// TwinCAT 3 PLC project Nestec
// libraries:
//   Tc2_ControllerToolbox,newest,Beckhoff Automation GmbH
//   Tc2_Standard,newest,Beckhoff Automation GmbH
//   Tc2_System,newest,Beckhoff Automation GmbH
//   Tc2_Utilities,newest,Beckhoff Automation GmbH
//   Tc3_Interfaces,3.3.0.0,Beckhoff Automation GmbH
//   Tc3_Module,3.3.6.0,Beckhoff Automation GmbH
// project tree:
//   Global Variables/ Global_Constantes.TcGVL, Global_IOs.TcGVL, TwinCAT_Configuration.TcGVL, Variable_Configuration.TcGVL
//   / GlobalImagePool.TcIPO (not stored), GlobalTextList.TcGTLO, Slow.TcTTO, Standard.TcTTO, Visualization Manager.TcVMO (not stored)
//   POUs/EMS/ EMS_Start.TcPOU
//   POUs/Flowrate management/ CALCULATE_FLOW.TcPOU, FLOWMETER.TcPOU
//   POUs/Functions/ PUMP_POWER.TcPOU, STATION_MODE.TcPOU
//   POUs/ MAIN.TcPOU
//   POUs/PC/ TO_PC.TcPOU
//   POUs/Tests/ getFlowrate.TcPOU, test.TcPOU, test_pressure.TcPOU, test_sonde_temp_G01.TcPOU, test_temp_G01.TcPOU, test_vacuum.TcPOU
//   Visualizations/ Visu1.TcVIS

CONFIGURATION Nestec
    RESOURCE PLC ON TwinCAT3
        TASK Slow(INTERVAL := T#100000us, PRIORITY := 21);
        TASK Standard(INTERVAL := T#10ms, PRIORITY := 20);
        PROGRAM CALCULATE_FLOW WITH Slow : CALCULATE_FLOW;
        PROGRAM MAIN WITH Standard : MAIN;
    END_RESOURCE
END_CONFIGURATION

// ---- Global Variables/Global_Constantes.TcGVL
{attribute 'Tc2GvlVarNames'}
VAR_GLOBAL


	R_BTN_S3: BOOL;



END_VAR

// ---- Global Variables/Global_IOs.TcGVL
{attribute 'Tc2GvlVarNames'}
VAR_GLOBAL

(**************************************
*
* PC variables 
*
***************************************)

(*FROM PC*)
	PC_ST1_PUMP_STATUS	:INT;(*0 OFF // 1 ON*)
	PC_ST2_PUMP_STATUS	:INT;
	PC_ST3_PUMP_STATUS	:INT;
	PC_ST4_PUMP_STATUS	:INT;

	PC_ST1_MODE			:INT;(*0 débit/pression // 1 pression max // 2 aspiration*)
	PC_ST2_MODE			:INT;
	PC_ST3_MODE			:INT;
	PC_ST4_MODE			:INT;

	PC_RESET_EMS			:BOOL; (*TO reset Emergency start*)

	PC_INIT					:BOOL;

(*TO PC*)
	PC_ST1_PRESSURE		:REAL;
	PC_ST2_PRESSURE		:REAL;
	PC_ST3_PRESSURE		:REAL;
	PC_ST4_PRESSURE		:REAL;

	PC_ST1_SUCTION		:REAL;
	PC_ST2_SUCTION		:REAL;
	PC_ST3_SUCTION		:REAL;
	PC_ST4_SUCTION		:REAL;

	PC_ST1_FLOWRATE		:REAL;
	PC_ST2_FLOWRATE		:REAL;
	PC_ST3_FLOWRATE		:REAL;
	PC_ST4_FLOWRATE		:REAL;

	PC_ST1_TEMP			:REAL;
	PC_ST2_TEMP			:REAL;
	PC_ST3_TEMP			:REAL;
	PC_ST4_TEMP			:REAL;

	PC_ST1_TEMP_ERROR	:BOOL;
	PC_ST2_TEMP_ERROR	:BOOL;
	PC_ST3_TEMP_ERROR	:BOOL;
	PC_ST4_TEMP_ERROR	:BOOL;

	PC_ST1_CURRENT		:REAL;
	PC_ST2_CURRENT		:REAL;
	PC_ST3_CURRENT		:REAL;
	PC_ST4_CURRENT		:REAL;

	PC_ST1_POWER			:REAL;
	PC_ST2_POWER			:REAL;
	PC_ST3_POWER			:REAL;
	PC_ST4_POWER			:REAL;

	PC_ST1_BTN			:BOOL;
	PC_ST2_BTN			:BOOL;
	PC_ST3_BTN			:BOOL;
	PC_ST4_BTN			:BOOL;

	PC_EMS_OK				:BOOL; (*EMS is SAFE*)






(**************************************
*
* EMERGECY STOP
*
***************************************)

	EMS_RESET		AT%Q*: BOOL;
	EMS_RUN		AT%Q*: BOOL;
	EMS_ACK 		AT%Q*: BOOL;

	EMS_FB_ERR	AT%I*: BOOL;
	EMS_COM_ERR	AT%I*: BOOL;
	EMS_OUT_ERR	AT%I*: BOOL;

	(*1: State RUN
	2: State STOP
	3: State SAFE
	4: State ERROR
	5: State RESET
	6: State START
	8: State DELAYOUT
	*)
	EMS_STATE		AT%I*:USINT;

	EMS_OK			AT%I*:BOOL;	(*Emergency stop is OK*)

(**************************************
*
* Inputs
*
***************************************)

	BTN_S3 AT%I*: BOOL;
	BTN_S4 AT%I*: BOOL;
	BTN_S5 AT%I*: BOOL;
	BTN_S6 AT%I*: BOOL;

	Weight_Station1 AT%I*:REAL;
	Weight_Station2 AT%I*:REAL;
	Weight_Station3 AT%I*:REAL;
	Weight_Station4 AT%I*:REAL;


	Temp_Station1 AT%I*:INT;
	Temp1_error   AT%I*:BOOL;
	Temp_Station2 AT%I*:INT;
	Temp2_error   AT%I*:BOOL;
	Temp_Station3 AT%I*:INT;
	Temp3_error   AT%I*:BOOL;
	Temp_Station4 AT%I*:INT;
	Temp4_error   AT%I*:BOOL;


	Vacuum_Station1 AT%I*:INT;
	Vacuum_Station2 AT%I*:INT;
	Vacuum_Station3 AT%I*:INT;
	Vacuum_Station4 AT%I*:INT;


	Pressure_Station1 AT%I*:INT;
	Pressure_Station2 AT%I*:INT;
	Pressure_Station3 AT%I*:INT;
	Pressure_Station4 AT%I*:INT;


	Temperature_entree_1 AT%I*:REAL;
	Temperature_entree_2 AT%I*:REAL;



(**************************************
*
* Outputs
*
***************************************)

	Alim_1 AT%Q*: BOOL;
	Alim_2 AT%Q*: BOOL;
	Alim_3 AT%Q*: BOOL;
	Alim_4 AT%Q*: BOOL;


	Mot_1 AT%Q*: BOOL;
	Mot_2 AT%Q*: BOOL;
	Mot_3 AT%Q*: BOOL;
	Mot_4 AT%Q*: BOOL;


	Solenoid_W13 AT%Q*: BOOL;
	Solenoid_W14 AT%Q*: BOOL;
	Solenoid_W15 AT%Q*: BOOL;
	Solenoid_W16 AT%Q*: BOOL;
	Solenoid_W17 AT%Q*: BOOL;
	Solenoid_W18 AT%Q*: BOOL;
	Solenoid_W19 AT%Q*: BOOL;
	Solenoid_W20 AT%Q*: BOOL;


	Light_H1 AT%Q*: BOOL;
	Light_H2 AT%Q*: BOOL;
	Light_H3 AT%Q*: BOOL;
	Light_H4 AT%Q*: BOOL;

(**************************************
*
* Multimeter IOs
*
***************************************)

	ST1_Multimeter_mode	AT%Q*:SINT := 3;
	ST2_Multimeter_mode	AT%Q*:SINT := 3;
	ST3_Multimeter_mode	AT%Q*:SINT := 3;
	ST4_Multimeter_mode	AT%Q*:SINT := 3;

(*
0 0x00 DC voltage
1 0x01 AC voltage
2 0x02 DC current
3 0x03 AC current
*)

	ST1_Multimeter_range AT%Q* :SINT := 1;
	ST2_Multimeter_range AT%Q* :SINT := 1;
	ST3_Multimeter_range AT%Q* :SINT := 1;
	ST4_Multimeter_range AT%Q* :SINT := 1;


(*
255 0xFF 300 mV / 100 mA
0 0x00  3 V / 1 A 
1 0x01 30 V / 10 A 
2 0x02 300 V (voltage only)  
*)


	ST1_Multimeter_value AT%I*:DINT;
	ST2_Multimeter_value AT%I*:DINT;
	ST3_Multimeter_value AT%I*:DINT;
	ST4_Multimeter_value AT%I*:DINT;



END_VAR

// ---- Global Variables/TwinCAT_Configuration.TcGVL
{attribute 'Tc2GvlVarNames'}
(* Generated automatically by TwinCAT - (read only) *)
VAR_CONFIG
	.EMS_RESET AT %QX8.0 : BOOL;	(*  ~ {LinkedWith:TIID^Device 2 (EtherCAT)^Armoire gauche (EK1100)^Term 13 (EL6900)^Module 2 (FSOE)^Standard In Vars RxPDO 1^Standard In Var 3} *)
	.EMS_RUN AT %QX12.0 : BOOL;	(*  ~ {LinkedWith:TIID^Device 2 (EtherCAT)^Armoire gauche (EK1100)^Term 13 (EL6900)^Module 2 (FSOE)^Standard In Vars RxPDO 1^Standard In Var 1} *)
	.EMS_ACK AT %QX12.1 : BOOL;	(*  ~ {LinkedWith:TIID^Device 2 (EtherCAT)^Armoire gauche (EK1100)^Term 13 (EL6900)^Module 2 (FSOE)^Standard In Vars RxPDO 1^Standard In Var 2} *)
	.EMS_FB_ERR AT %IX76.0 : BOOL;	(*  ~ {LinkedWith:TIID^Device 2 (EtherCAT)^Armoire gauche (EK1100)^Term 13 (EL6900)^Module 2 (FSOE)^Standard Out Vars TxPDO 1^Standard Out Var 1} *)
	.EMS_COM_ERR AT %IX76.1 : BOOL;	(*  ~ {LinkedWith:TIID^Device 2 (EtherCAT)^Armoire gauche (EK1100)^Term 13 (EL6900)^Module 2 (FSOE)^Standard Out Vars TxPDO 1^Standard Out Var 2} *)
	.EMS_OUT_ERR AT %IX76.2 : BOOL;	(*  ~ {LinkedWith:TIID^Device 2 (EtherCAT)^Armoire gauche (EK1100)^Term 13 (EL6900)^Module 2 (FSOE)^Standard Out Vars TxPDO 1^Standard Out Var 3} *)
	.EMS_STATE AT %IB92 : USINT;	(*  ~ {LinkedWith:TIID^Device 2 (EtherCAT)^Armoire gauche (EK1100)^Term 13 (EL6900)^Module 2 (FSOE)^FB Info Data^Info FB 1^State} *)
	.EMS_OK AT %IX88.0 : BOOL;	(*  ~ {LinkedWith:TIID^Device 2 (EtherCAT)^Armoire gauche (EK1100)^Term 13 (EL6900)^Module 2 (FSOE)^Standard Out Vars TxPDO 1^Standard Out Var 4} *)
	.BTN_S3 AT %IX56.0 : BOOL;	(*  ~ {LinkedWith:TIID^Device 2 (EtherCAT)^Armoire gauche (EK1100)^Term 24 (EL1002)^Channel 1^S3} *)
	.BTN_S4 AT %IX56.1 : BOOL;	(*  ~ {LinkedWith:TIID^Device 2 (EtherCAT)^Armoire gauche (EK1100)^Term 25 (EL1002)^Channel 1^S4} *)
	.BTN_S5 AT %IX56.2 : BOOL;	(*  ~ {LinkedWith:TIID^Device 2 (EtherCAT)^Armoire droite (EK1100)^Term 41 (EL1002)^Channel 1^S5} *)
	.BTN_S6 AT %IX56.3 : BOOL;	(*  ~ {LinkedWith:TIID^Device 2 (EtherCAT)^Armoire droite (EK1100)^Term 42 (EL1002)^Channel 1^S6} *)
	.Weight_Station1 AT %IB96 : REAL;	(*  ~ {LinkedWith:TIID^Device 2 (EtherCAT)^Armoire gauche (EK1100)^Term 9 (EL3356-0010)^RMB Value (Real)^Value (Real)} *)
	.Weight_Station2 AT %IB100 : REAL;	(*  ~ {LinkedWith:TIID^Device 2 (EtherCAT)^Armoire gauche (EK1100)^Term 10 (EL3356-0010)^RMB Value (Real)^Value (Real)} *)
	.Weight_Station3 AT %IB104 : REAL;	(*  ~ {LinkedWith:TIID^Device 2 (EtherCAT)^Armoire droite (EK1100)^Term 58 (EL3356-0010)^RMB Value (Real)^Value (Real)} *)
	.Weight_Station4 AT %IB108 : REAL;	(*  ~ {LinkedWith:TIID^Device 2 (EtherCAT)^Armoire droite (EK1100)^Term 59 (EL3356-0010)^RMB Value (Real)^Value (Real)} *)
	.Temp_Station1 AT %IB16 : INT;	(*  ~ {LinkedWith:TIID^Device 2 (EtherCAT)^Armoire gauche (EK1100)^Term 11 (EL3312)^TC Inputs Channel 1^Value} *)
	.Temp1_error AT %IX56.4 : BOOL;	(*  ~ {LinkedWith:TIID^Device 2 (EtherCAT)^Armoire gauche (EK1100)^Term 11 (EL3312)^TC Inputs Channel 1^Status^Error} *)
	.Temp_Station2 AT %IB18 : INT;	(*  ~ {LinkedWith:TIID^Device 2 (EtherCAT)^Armoire gauche (EK1100)^Term 11 (EL3312)^TC Inputs Channel 2^Value} *)
	.Temp2_error AT %IX56.5 : BOOL;	(*  ~ {LinkedWith:TIID^Device 2 (EtherCAT)^Armoire gauche (EK1100)^Term 11 (EL3312)^TC Inputs Channel 2^Status^Error} *)
	.Temp_Station3 AT %IB20 : INT;	(*  ~ {LinkedWith:TIID^Device 2 (EtherCAT)^Armoire droite (EK1100)^Term 60 (EL3312)^TC Inputs Channel 1^Value} *)
	.Temp3_error AT %IX56.6 : BOOL;
	.Temp_Station4 AT %IB22 : INT;	(*  ~ {LinkedWith:TIID^Device 2 (EtherCAT)^Armoire droite (EK1100)^Term 60 (EL3312)^TC Inputs Channel 2^Value} *)
	.Temp4_error AT %IX56.7 : BOOL;
	.Vacuum_Station1 AT %IB60 : INT;	(*  ~ {LinkedWith:TIID^Device 2 (EtherCAT)^Armoire gauche (EK1100)^Term 12 (EL3054)^AI Standard Channel 1^Value_Suction_Poste1} *)
	.Vacuum_Station2 AT %IB62 : INT;	(*  ~ {LinkedWith:TIID^Device 2 (EtherCAT)^Armoire gauche (EK1100)^Term 12 (EL3054)^AI Standard Channel 2^Value_Suction_Poste2} *)
	.Vacuum_Station3 AT %IB64 : INT;	(*  ~ {LinkedWith:TIID^Device 2 (EtherCAT)^Armoire droite (EK1100)^Term 62 (EL3054)^AI Standard Channel 1^Value_Suction_Poste3} *)
	.Vacuum_Station4 AT %IB66 : INT;	(*  ~ {LinkedWith:TIID^Device 2 (EtherCAT)^Armoire droite (EK1100)^Term 62 (EL3054)^AI Standard Channel 2^Value_Suction_Poste4} *)
	.Pressure_Station1 AT %IB68 : INT;	(*  ~ {LinkedWith:TIID^Device 2 (EtherCAT)^Armoire gauche (EK1100)^Term 12 (EL3054)^AI Standard Channel 3^Value_Pressure_Poste1} *)
	.Pressure_Station2 AT %IB70 : INT;	(*  ~ {LinkedWith:TIID^Device 2 (EtherCAT)^Armoire gauche (EK1100)^Term 12 (EL3054)^AI Standard Channel 4^Value_Pressure_Poste2} *)
	.Pressure_Station3 AT %IB72 : INT;	(*  ~ {LinkedWith:TIID^Device 2 (EtherCAT)^Armoire droite (EK1100)^Term 62 (EL3054)^AI Standard Channel 3^Value_Pressure_Poste3} *)
	.Pressure_Station4 AT %IB74 : INT;	(*  ~ {LinkedWith:TIID^Device 2 (EtherCAT)^Armoire droite (EK1100)^Term 62 (EL3054)^AI Standard Channel 4^Value_Pressure_Poste4} *)
	.Temperature_entree_1 AT %IB80 : REAL;
	.Temperature_entree_2 AT %IB84 : REAL;
	.Alim_1 AT %QX4.0 : BOOL;	(*  ~ {LinkedWith:TIID^Device 2 (EtherCAT)^Armoire gauche (EK1100)^Term 16 (EL2622)^Channel 1^Output_L_Alim1;TIID^Device 2 (EtherCAT)^Armoire gauche (EK1100)^Term 16 (EL2622)^Channel 2^Output_N_Alim1} *)
	.Alim_2 AT %QX4.1 : BOOL;	(*  ~ {LinkedWith:TIID^Device 2 (EtherCAT)^Armoire gauche (EK1100)^Term 17 (EL2622)^Channel 1^Output_L_Alim2;TIID^Device 2 (EtherCAT)^Armoire gauche (EK1100)^Term 17 (EL2622)^Channel 2^Output_N_Alim2} *)
	.Alim_3 AT %QX4.2 : BOOL;	(*  ~ {LinkedWith:TIID^Device 2 (EtherCAT)^Armoire droite (EK1100)^Term 63 (EL2622)^Channel 1^Output_L_Alim3;TIID^Device 2 (EtherCAT)^Armoire droite (EK1100)^Term 63 (EL2622)^Channel 2^Output_N_Alim3} *)
	.Alim_4 AT %QX4.3 : BOOL;	(*  ~ {LinkedWith:TIID^Device 2 (EtherCAT)^Armoire droite (EK1100)^Term 65 (EL2622)^Channel 1^Output_L_Alim4;TIID^Device 2 (EtherCAT)^Armoire droite (EK1100)^Term 65 (EL2622)^Channel 2^Output_N_Alim4} *)
	.Mot_1 AT %QX4.4 : BOOL;	(*  ~ {LinkedWith:TIID^Device 2 (EtherCAT)^Armoire gauche (EK1100)^Term 18 (EL2622)^Channel 1^Output_L_Mot1;TIID^Device 2 (EtherCAT)^Armoire gauche (EK1100)^Term 18 (EL2622)^Channel 2^Output_N_Mot1} *)
	.Mot_2 AT %QX4.5 : BOOL;	(*  ~ {LinkedWith:TIID^Device 2 (EtherCAT)^Armoire gauche (EK1100)^Term 19 (EL2622)^Channel 1^Output_L_Mot2;TIID^Device 2 (EtherCAT)^Armoire gauche (EK1100)^Term 19 (EL2622)^Channel 2^Output_N_Mot2} *)
	.Mot_3 AT %QX4.6 : BOOL;	(*  ~ {LinkedWith:TIID^Device 2 (EtherCAT)^Armoire droite (EK1100)^Term 64 (EL2622)^Channel 1^Output_L_Mot3;TIID^Device 2 (EtherCAT)^Armoire droite (EK1100)^Term 64 (EL2622)^Channel 2^Output_N_Mot3} *)
	.Mot_4 AT %QX4.7 : BOOL;	(*  ~ {LinkedWith:TIID^Device 2 (EtherCAT)^Armoire droite (EK1100)^Term 66 (EL2622)^Channel 1^Output_L_Mot4;TIID^Device 2 (EtherCAT)^Armoire droite (EK1100)^Term 66 (EL2622)^Channel 2^Output_N_Mot4} *)
	.Solenoid_W13 AT %QX0.0 : BOOL;	(*  ~ {LinkedWith:TIID^Device 2 (EtherCAT)^Armoire gauche (EK1100)^Term 27 (EL2002)^Channel 1^W13} *)
	.Solenoid_W14 AT %QX0.1 : BOOL;	(*  ~ {LinkedWith:TIID^Device 2 (EtherCAT)^Armoire gauche (EK1100)^Term 27 (EL2002)^Channel 2^W14} *)
	.Solenoid_W15 AT %QX0.2 : BOOL;	(*  ~ {LinkedWith:TIID^Device 2 (EtherCAT)^Armoire gauche (EK1100)^Term 28 (EL2002)^Channel 1^W15} *)
	.Solenoid_W16 AT %QX0.3 : BOOL;	(*  ~ {LinkedWith:TIID^Device 2 (EtherCAT)^Armoire gauche (EK1100)^Term 28 (EL2002)^Channel 2^W16} *)
	.Solenoid_W17 AT %QX0.4 : BOOL;	(*  ~ {LinkedWith:TIID^Device 2 (EtherCAT)^Armoire droite (EK1100)^Term 44 (EL2002)^Channel 1^W17} *)
	.Solenoid_W18 AT %QX0.5 : BOOL;	(*  ~ {LinkedWith:TIID^Device 2 (EtherCAT)^Armoire droite (EK1100)^Term 44 (EL2002)^Channel 2^W18} *)
	.Solenoid_W19 AT %QX0.6 : BOOL;	(*  ~ {LinkedWith:TIID^Device 2 (EtherCAT)^Armoire droite (EK1100)^Term 45 (EL2002)^Channel 1^W19} *)
	.Solenoid_W20 AT %QX0.7 : BOOL;	(*  ~ {LinkedWith:TIID^Device 2 (EtherCAT)^Armoire droite (EK1100)^Term 45 (EL2002)^Channel 2^W20} *)
	.Light_H1 AT %QX1.0 : BOOL;	(*  ~ {LinkedWith:TIID^Device 2 (EtherCAT)^Armoire gauche (EK1100)^Term 32 (EL2004)^Channel 1^H1} *)
	.Light_H2 AT %QX1.1 : BOOL;	(*  ~ {LinkedWith:TIID^Device 2 (EtherCAT)^Armoire gauche (EK1100)^Term 32 (EL2004)^Channel 3^H2} *)
	.Light_H3 AT %QX1.2 : BOOL;	(*  ~ {LinkedWith:TIID^Device 2 (EtherCAT)^Armoire droite (EK1100)^Term 46 (EL2004)^Channel 1^H3} *)
	.Light_H4 AT %QX1.3 : BOOL;	(*  ~ {LinkedWith:TIID^Device 2 (EtherCAT)^Armoire droite (EK1100)^Term 46 (EL2004)^Channel 3^H4} *)
	.ST1_Multimeter_mode AT %QB16 : SINT;	(*  ~ {LinkedWith:TIID^Device 2 (EtherCAT)^Armoire gauche (EK1100)^Term 39 (EL3681)^SAI Range^Control^Mode} *)
	.ST2_Multimeter_mode AT %QB20 : SINT;
	.ST3_Multimeter_mode AT %QB21 : SINT;
	.ST4_Multimeter_mode AT %QB22 : SINT;
	.ST1_Multimeter_range AT %QB17 : SINT;	(*  ~ {LinkedWith:TIID^Device 2 (EtherCAT)^Armoire gauche (EK1100)^Term 39 (EL3681)^SAI Range^Control^Range} *)
	.ST2_Multimeter_range AT %QB23 : SINT;
	.ST3_Multimeter_range AT %QB24 : SINT;
	.ST4_Multimeter_range AT %QB25 : SINT;
	.ST1_Multimeter_value AT %IB112 : DINT;	(*  ~ {LinkedWith:TIID^Device 2 (EtherCAT)^Armoire gauche (EK1100)^Term 39 (EL3681)^SAI Inputs^Value} *)
	.ST2_Multimeter_value AT %IB116 : DINT;
	.ST3_Multimeter_value AT %IB120 : DINT;
	.ST4_Multimeter_value AT %IB124 : DINT;
END_VAR

// ---- Global Variables/Variable_Configuration.TcGVL
{attribute 'Tc2GvlVarNames'}
VAR_CONFIG
END_VAR

// ---- POUs/Flowrate management/CALCULATE_FLOW.TcPOU
PROGRAM CALCULATE_FLOW

VAR

	FLOW		:REAL;
	POIDS_1_OLD: REAL;
	FLOW_1: REAL;

	FB_CTRL_PT3_POIDS_1: FB_CTRL_PT3;

	eMode_POIDS_1: E_CTRL_MODE;
	stParams_POIDS_1: ST_CTRL_PT3_PARAMS;

	POIDS_1_FILTERED: REAL;
	FLOW_1_FILTERED: REAL;
	POIDS_1_FILTERED_OLD: REAL;
	FLOW_2: REAL;
	FLOW_3: REAL;
	FLOW_4: REAL;
	POIDS_2_OLD: REAL;
	POIDS_3_OLD: REAL;
	POIDS_4_OLD: REAL;
	FLOW_2_FILTERED: REAL;
	FLOW_3_FILTERED: REAL;
	FLOW_4_FILTERED: REAL;
	POIDS_2_FILTERED: REAL;
	POIDS_3_FILTERED: REAL;
	POIDS_4_FILTERED: REAL;
	POIDS_2_FILTERED_OLD: REAL;
	POIDS_3_FILTERED_OLD: REAL;
	POIDS_4_FILTERED_OLD: REAL;
	FB_CTRL_PT3_POIDS_2:  FB_CTRL_PT3;
	FB_CTRL_PT3_POIDS_3:  FB_CTRL_PT3;
	FB_CTRL_PT3_POIDS_4:  FB_CTRL_PT3;
END_VAR

(*PARAMETRES FILTRES*)

	(* init parameter struct *)
	stParams_POIDS_1.tCtrlCycleTime			:= T#100ms;
	stParams_POIDS_1.tTaskCycleTime			:= T#100ms;
	stParams_POIDS_1.tT1					:= T#1s000ms;
	stParams_POIDS_1.tT2					:= T#1s000ms;
	stParams_POIDS_1.tT3					:= T#1s000ms;
	stParams_POIDS_1.fKp					:= 1;

	(* set the mode to ACTIVE --> normal operation *)
	eMode_POIDS_1							:= eCTRL_MODE_ACTIVE;


(*calcule du débit en fonction de la différence de poids*)
FLOW_1 := (Weight_Station1-POIDS_1_OLD)*600;
FLOW_2 := (Weight_Station2-POIDS_2_OLD)*600;
FLOW_3 := (Weight_Station3-POIDS_3_OLD)*600;
FLOW_4 := (Weight_Station4-POIDS_4_OLD)*600;



(*Filtres 3 ème ordre*)
FB_CTRL_PT3_POIDS_1(
	fIn:= Weight_Station1,
	fManValue:= 0,
	eMode:= eMode_POIDS_1,
	bHold:= FALSE ,
	stParams:= stParams_POIDS_1,
	fOut=> POIDS_1_FILTERED );
FB_CTRL_PT3_POIDS_2(
	fIn:= Weight_Station2,
	fManValue:= 0,
	eMode:= eMode_POIDS_1,
	bHold:= FALSE ,
	stParams:= stParams_POIDS_1,
	fOut=> POIDS_2_FILTERED );
FB_CTRL_PT3_POIDS_3(
	fIn:= Weight_Station3,
	fManValue:= 0,
	eMode:= eMode_POIDS_1,
	bHold:= FALSE ,
	stParams:= stParams_POIDS_1,
	fOut=> POIDS_3_FILTERED );
FB_CTRL_PT3_POIDS_4(
	fIn:= Weight_Station4,
	fManValue:= 0,
	eMode:= eMode_POIDS_1,
	bHold:= FALSE ,
	stParams:= stParams_POIDS_1,
	fOut=> POIDS_4_FILTERED );

FLOW_1_FILTERED := (POIDS_1_FILTERED-POIDS_1_FILTERED_OLD)*600;
FLOW_2_FILTERED := (POIDS_2_FILTERED-POIDS_2_FILTERED_OLD)*600;
FLOW_3_FILTERED := (POIDS_3_FILTERED-POIDS_3_FILTERED_OLD)*600;
FLOW_4_FILTERED := (POIDS_4_FILTERED-POIDS_4_FILTERED_OLD)*600;




POIDS_1_OLD := Weight_Station1;
POIDS_2_OLD := Weight_Station2;
POIDS_3_OLD := Weight_Station3;
POIDS_4_OLD := Weight_Station4;

POIDS_1_FILTERED_OLD:=POIDS_1_FILTERED;
POIDS_2_FILTERED_OLD:=POIDS_2_FILTERED;
POIDS_3_FILTERED_OLD:=POIDS_3_FILTERED;
POIDS_4_FILTERED_OLD:=POIDS_4_FILTERED;

END_PROGRAM

// ---- POUs/MAIN.TcPOU
PROGRAM MAIN
VAR

	STATION_MODE_ST1: STATION_MODE;
	PUMP_POWER_ST1: PUMP_POWER;
	FLOWMETER_ST1: FLOWMETER;



	FLOWMETER_ST4: FLOWMETER;
	FLOWMETER_ST3: FLOWMETER;
	FLOWMETER_ST2: FLOWMETER;
	STATION_MODE_ST2: STATION_MODE;
	STATION_MODE_ST3: STATION_MODE;
	STATION_MODE_ST4: STATION_MODE;
	PUMP_POWER_ST2: PUMP_POWER;
	PUMP_POWER_ST3: PUMP_POWER;
	PUMP_POWER_ST4: PUMP_POWER;
END_VAR

(******************************************************
*
* Test
*
****************************************************)


(******************************************************
*
* Emergency tread
*
****************************************************)

EMS_Start();

(*****************************************************
*
* Stations
*
*******************************************************)
(* gestion des électrovannes*)
STATION_MODE_ST1(
	mode:= PC_ST1_MODE,
	vacuum_valve=>Solenoid_W13 ,
	pressure_valve=>Solenoid_W14 );
STATION_MODE_ST2(
	mode:= PC_ST2_MODE,
	vacuum_valve=>Solenoid_W15 ,
	pressure_valve=>Solenoid_W16 );
STATION_MODE_ST3(
	mode:= PC_ST3_MODE,
	vacuum_valve=>Solenoid_W17,
	pressure_valve=>Solenoid_W18 );
STATION_MODE_ST4(
	mode:= PC_ST4_MODE,
	vacuum_valve=>Solenoid_W19 ,
	pressure_valve=>Solenoid_W20 );

(*gestion de l'alimentation des pompes*)
PUMP_POWER_ST1(
	PUMP_STATUS:= PC_ST1_PUMP_STATUS,
	EMS_OK:= EMS_OK,
	POWER=> Alim_1,
	POWER_LED=> Light_H1);
PUMP_POWER_ST2(
	PUMP_STATUS:= PC_ST2_PUMP_STATUS,
	EMS_OK:= EMS_OK,
	POWER=> Alim_2,
	POWER_LED=> Light_H2);
PUMP_POWER_ST3(
	PUMP_STATUS:= PC_ST3_PUMP_STATUS,
	EMS_OK:= EMS_OK,
	POWER=> Alim_3,
	POWER_LED=> Light_H3);
PUMP_POWER_ST4(
	PUMP_STATUS:= PC_ST4_PUMP_STATUS,
	EMS_OK:= EMS_OK,
	POWER=> Alim_4,
	POWER_LED=> Light_H4);

(* FLOWMETER *)
FLOWMETER_ST1(
	ON:= TRUE,
	POIDS			:= Weight_Station1,
	POIDS_BAS		:= 900,
	POIDS_HAUT	:= 2300,
	PC_MODE 		:= PC_ST1_MODE,
	FLOWRATE		:=CALCULATE_FLOW.FLOW_1_FILTERED,
	DEBIT			=> PC_ST1_FLOWRATE,
	PURGE			=> Mot_1);
FLOWMETER_ST2(
	ON:= TRUE,
	POIDS			:= Weight_Station2,
	POIDS_BAS		:= 800,
	POIDS_HAUT	:= 2100,
	PC_MODE 		:= PC_ST2_MODE,
	FLOWRATE		:=CALCULATE_FLOW.FLOW_2_FILTERED,
	DEBIT			=> PC_ST2_FLOWRATE,
	PURGE			=> Mot_2);
FLOWMETER_ST3(
	ON:= TRUE,
	POIDS			:= Weight_Station3,
	POIDS_BAS		:= 1200,
	POIDS_HAUT	:= 2300,
	PC_MODE 		:= PC_ST3_MODE,
	FLOWRATE		:=CALCULATE_FLOW.FLOW_3_FILTERED,
	DEBIT			=> PC_ST3_FLOWRATE,
	PURGE			=> Mot_3);
FLOWMETER_ST4(
	ON:= TRUE,
	POIDS			:= Weight_Station4,
	POIDS_BAS		:= 1000,
	POIDS_HAUT	:= 2300,
	PC_MODE 		:= PC_ST4_MODE,
	FLOWRATE		:=CALCULATE_FLOW.FLOW_4_FILTERED,
	DEBIT			=> PC_ST4_FLOWRATE,
	PURGE			=> Mot_4);

(*****************************************************
*
* PC tread
*
*******************************************************)
TO_PC();

END_PROGRAM

// ---- POUs/Functions/STATION_MODE.TcPOU
FUNCTION_BLOCK STATION_MODE

VAR_INPUT
	mode :INT;
END_VAR

VAR_OUTPUT
	vacuum_valve 	:BOOL;
	pressure_valve	:BOOL;
END_VAR

VAR

END_VAR



CASE mode OF

0:(*Débit*)
vacuum_valve	:= 	TRUE;
pressure_valve	:=	TRUE;

1:(*Pmax*)
vacuum_valve	:= 	TRUE;
pressure_valve	:=	FALSE;

2:(*Aspiration*)
vacuum_valve	:= 	FALSE;
pressure_valve	:=	TRUE;

ELSE

vacuum_valve	:= 	FALSE;
pressure_valve	:=	FALSE;

END_CASE;

END_FUNCTION_BLOCK

// ---- POUs/Functions/PUMP_POWER.TcPOU
FUNCTION_BLOCK PUMP_POWER

VAR_INPUT
	PUMP_STATUS	:INT;
	EMS_OK			:BOOL;
END_VAR

VAR_OUTPUT
	POWER			:BOOL;
	POWER_LED	:BOOL;
END_VAR

VAR
END_VAR

IF PUMP_STATUS=1 AND EMS_OK THEN

POWER:=TRUE;
POWER_LED:=TRUE;

ELSE

POWER:=FALSE;
POWER_LED:=FALSE;

END_IF;

END_FUNCTION_BLOCK

// ---- POUs/Flowrate management/FLOWMETER.TcPOU
FUNCTION_BLOCK FLOWMETER

(***************************************
-1 	-> purge
-99 	-> OFF
xxx	-> en cours de mesure
***************************************)

VAR_INPUT

	ON				:BOOL; (*active/desactive la gestion du débit/purge*)
	POIDS			:REAL; (*poids actuel*)
	POIDS_BAS		:REAL; (*en grammes / Limite bas*)
	POIDS_HAUT	:REAL; (*limite haut*)
	FLOWRATE		:REAL; (*débit instantané*)
	PC_MODE		:INT; (*mode de la station*)

END_VAR

VAR_OUTPUT

	DEBIT			:REAL; (*Valeur du débit en ml/min*)
	PURGE			:BOOL; (*commande de la pompe de vidange*)

END_VAR

VAR
END_VAR

IF ON=TRUE THEN

	IF (POIDS < POIDS_HAUT) AND NOT PURGE AND  PC_MODE=0 THEN

		(*calcule ici le débit*)
		IF FLOWRATE > 10 THEN
			DEBIT:=FLOWRATE;
		ELSE
			DEBIT:=0;
		END_IF;

	ELSIF POIDS < POIDS_BAS THEN

		PURGE:=FALSE;

	ELSIF  (POIDS > POIDS_HAUT) OR PC_MODE<>0  THEN

		PURGE:=TRUE;
		DEBIT:=-1; (*-1 indique la purge*)


	END_IF;


ELSE

PURGE:=FALSE;
DEBIT:=-99.0;

END_IF;

END_FUNCTION_BLOCK

// ---- POUs/EMS/EMS_Start.TcPOU
PROGRAM EMS_Start
VAR
	RESET: BOOL;
END_VAR

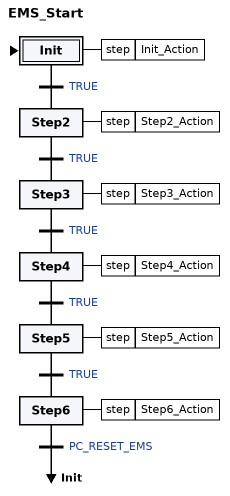
INITIAL_STEP Init:
    Init_Action(N);  // step action
END_STEP
TRANSITION FROM Init TO Step2
    := TRUE;
END_TRANSITION
STEP Step2:
    Step2_Action(N);  // step action
END_STEP
TRANSITION FROM Step2 TO Step3
    := TRUE;
END_TRANSITION
STEP Step3:  // min time t#1s
    Step3_Action(N);  // step action
END_STEP
TRANSITION FROM Step3 TO Step4
    := TRUE;
END_TRANSITION
STEP Step4:
    Step4_Action(N);  // step action
END_STEP
TRANSITION FROM Step4 TO Step5
    := TRUE;
END_TRANSITION
STEP Step5:  // min time t#1s
    Step5_Action(N);  // step action
END_STEP
TRANSITION FROM Step5 TO Step6
    := TRUE;
END_TRANSITION
STEP Step6:
    Step6_Action(N);  // step action
END_STEP
TRANSITION FROM Step6 TO Init
    := PC_RESET_EMS;
END_TRANSITION

ACTION Step6_Action:
EMS_RESET:=FALSE;
END_ACTION

ACTION Init_Action:

	EMS_RUN:=FALSE;
	EMS_ACK:=FALSE;
	EMS_RESET:=FALSE;

	RESET:=FALSE;
END_ACTION

ACTION Step3_Action:
EMS_ACK:=TRUE;
END_ACTION

ACTION Step4_Action:
EMS_ACK:=FALSE;
END_ACTION

ACTION Step2_Action:
EMS_RUN:=TRUE;
END_ACTION

ACTION Step5_Action:
EMS_RESET:=TRUE;
END_ACTION

END_PROGRAM

// ---- POUs/PC/TO_PC.TcPOU
PROGRAM TO_PC
VAR

	R_TRIG_S3: R_TRIG;


	R_TRIG_S4: R_TRIG;
	R_TRIG_S5: R_TRIG;
	R_TRIG_S6: R_TRIG;
	R_BTN_S4: BOOL;
	R_BTN_S6: BOOL;
	R_BTN_S5: BOOL;
END_VAR

(*TO PC*)

	PC_ST1_PRESSURE:=Pressure_Station1/32767.0*25.0+0.05;
	PC_ST2_PRESSURE:=(Pressure_Station2-190)/32767.0*25.0;
	PC_ST3_PRESSURE:=(Pressure_Station3-25)/32767.0*25.0;
	PC_ST4_PRESSURE:=Pressure_Station4/32767.0*25.0+0.05;

	PC_ST1_SUCTION:=Vacuum_Station1/32767.0*4.0-1.0;
	PC_ST2_SUCTION:=Vacuum_Station2/32767.0*4.0-1.0;
	PC_ST3_SUCTION:=Vacuum_Station3/32767.0*4.0-1.0;
	PC_ST4_SUCTION:=Vacuum_Station4/32767.0*4.0-1.0;

	PC_ST1_FLOWRATE:=MAIN.FLOWMETER_ST1.DEBIT;
	PC_ST2_FLOWRATE:=MAIN.FLOWMETER_ST2.DEBIT;
	PC_ST3_FLOWRATE:=MAIN.FLOWMETER_ST3.DEBIT;
	PC_ST4_FLOWRATE:=MAIN.FLOWMETER_ST4.DEBIT;

	PC_ST1_TEMP:=Temp_Station1/10.0;
	PC_ST2_TEMP:=Temp_Station2/10.0;
	PC_ST3_TEMP:=Temp_Station3/10.0;
	PC_ST4_TEMP:=Temp_Station4/10.0;

	PC_ST1_TEMP_ERROR	:=Temp1_error; (*TRUE IF AN ERROR OCCURE / THE SENSOR IS NOT CONNECTED*)
	PC_ST2_TEMP_ERROR	:=Temp2_error;
	PC_ST3_TEMP_ERROR	:=Temp3_error;
	PC_ST4_TEMP_ERROR	:=Temp4_error;

	PC_ST1_CURRENT := ST1_Multimeter_value/1000.0/1000.0;(*représentation en Ampères*)
	PC_ST2_CURRENT := ST2_Multimeter_value/1000.0/1000.0;;
	PC_ST3_CURRENT := ST3_Multimeter_value/1000.0/1000.0;;
	PC_ST4_CURRENT := ST4_Multimeter_value/1000.0/1000.0;;

	PC_ST1_POWER;
	PC_ST2_POWER;
	PC_ST3_POWER;
	PC_ST4_POWER;

(*GESTION BOUTONS*)

IF R_BTN_S3 AND PC_ST1_BTN=0 THEN
PC_ST1_BTN:=1;
ELSIF R_BTN_S3 AND PC_ST1_BTN=1 THEN
PC_ST1_BTN:=0;
END_IF

IF R_BTN_S4 AND PC_ST2_BTN=0 THEN
PC_ST2_BTN:=1;
ELSIF R_BTN_S4 AND PC_ST2_BTN=1 THEN
PC_ST2_BTN:=0;
END_IF

IF R_BTN_S5 AND PC_ST3_BTN=0 THEN
PC_ST3_BTN:=1;
ELSIF R_BTN_S5 AND PC_ST3_BTN=1 THEN
PC_ST3_BTN:=0;
END_IF

IF R_BTN_S6 AND PC_ST4_BTN=0 THEN
PC_ST4_BTN:=1;
ELSIF R_BTN_S6 AND PC_ST4_BTN=1 THEN
PC_ST4_BTN:=0;
END_IF

	PC_EMS_OK			:=EMS_OK;


(*****************************************************
*
* PC INIT
*
*******************************************************)
IF PC_INIT THEN
PC_ST1_BTN:=FALSE;
PC_ST2_BTN:=FALSE;
PC_ST3_BTN:=FALSE;
PC_ST4_BTN:=FALSE;
END_IF;

(*****************************************************
*
* Edges Detections
*
*******************************************************)
R_TRIG_S3(CLK:= BTN_S3, Q=> R_BTN_S3);
R_TRIG_S4(CLK:= BTN_S4, Q=> R_BTN_S4);
R_TRIG_S5(CLK:= BTN_S5, Q=> R_BTN_S5);
R_TRIG_S6(CLK:= BTN_S6, Q=> R_BTN_S6);

END_PROGRAM

// ---- POUs/Tests/getFlowrate.TcPOU
PROGRAM getFlowrate
VAR

	flowrate: LREAL;
	poids_old: REAL;

END_VAR



VAR

END_VAR



flowrate := (Weight_Station1-poids_old)/20*3600/1000.0/1000.0;

poids_old := Weight_Station1;




flowrate := (Weight_Station2-poids_old)/20*3600/1000.0/1000.0;

poids_old := Weight_Station2;




flowrate := (Weight_Station3-poids_old)/20*3600/1000.0/1000.0;

poids_old := Weight_Station3;





flowrate := (Weight_Station4-poids_old)/20*3600/1000.0/1000.0;

poids_old := Weight_Station4;

END_PROGRAM

// ---- POUs/Tests/test.TcPOU
PROGRAM test
VAR
	TP_BTN1: TP;
END_VAR



TP_BTN1(IN:= BTN_S3, PT:= t#3s, Q=> Light_H1);

Light_H2 := (TP_BTN1.ET > t#1s) AND (TP_BTN1.ET < t#2s);

END_PROGRAM

// ---- POUs/Tests/test_pressure.TcPOU
 PROGRAM test_pressure


VAR
	Pressure_post1:REAL;
	Pressure_post2:REAL;
	Pressure_post3:REAL;
	Pressure_post4:REAL;

END_VAR


Pressure_post1:= (Pressure_Station1 - 4.0)* 24.7/16.0/2000.0;
Pressure_post2:= (Pressure_Station2 - 4.0)* 24.0/16.0/2000.0;
Pressure_post3:= (Pressure_Station3 - 4.0)* 24.2/16.0/2000.0;
Pressure_post4:= (Pressure_Station4 - 4.0)* 24.7/16.0/2000.0;

END_PROGRAM

// ---- POUs/Tests/test_sonde_temp_G01.TcPOU
PROGRAM test_sonde_temp_G01


VAR

	Temp_St1: REAL;
	Temp_St2: REAL;

END_VAR





Temp_St1:= (-30.76) * LN(Temperature_entree_1) + 308.76;
Temp_St2:= (-30.76) * LN(Temperature_entree_2) + 308.76;

END_PROGRAM

// ---- POUs/Tests/test_temp_G01.TcPOU
PROGRAM test_temp_G01

VAR
	Temperature_G01_1:REAL;
	Temperature_G01_2:REAL;
	Temperature_G01_3:REAL;
	Temperature_G01_4:REAL;

END_VAR



Temperature_G01_1:= Temp_Station1/10.0;
Temperature_G01_2:= Temp_Station2/10.0;
Temperature_G01_3:= Temp_Station3/10.0;
Temperature_G01_4:= Temp_Station4/10.0;

IF Temp1_error=TRUE THEN

Temperature_G01_1:=-9999;

END_IF

END_PROGRAM

// ---- POUs/Tests/test_vacuum.TcPOU
PROGRAM test_vacuum

VAR
	Vacuum_post1:REAL;
	Vacuum_post2:REAL;
	Vacuum_post3:REAL;
	Vacuum_post4:REAL;

END_VAR



Vacuum_post1:= ((Vacuum_Station1 - 8.0)* 3.8/16.0/2000)-1;
Vacuum_post2:= ((Vacuum_Station2 - 8.0)* 4.0/16.0/2000)-1;
Vacuum_post3:= ((Vacuum_Station3 - 8.0)* 4.0/16.0/2000)-1;
Vacuum_post4:= ((Vacuum_Station4 - 8.0)* 4.0/16.0/2000)-1;

END_PROGRAM

// ---- Visualizations/Visu1.TcVIS
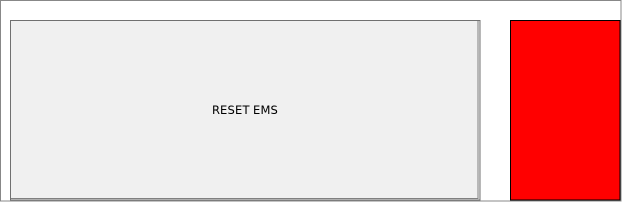
VISUALIZATION Visu1  // 622x202
    Button (10,20 470x180), "RESET EMS"
        tap Global_IOs.PC_RESET_EMS
    Rectangle (510,20 110x180), colour toggle: Global_IOs.EMS_OK
END_VISUALIZATION
